KUKA KRL data list: ITEMPICK_ADDRETURN.dat

&ACCESS RVP
&REL 1
&PARAM EDITMASK = *
DEFDAT ITEMPICK_ADDRETURN
ENDDAT
